
FUNCTION CB_dint_to_dword : DWORD

TITLE = ' Convert a double integer into an Dword '
VERSION : '1.0'
AUTHOR  : CB
NAME    : DinToDwo
FAMILY  : TNI

VAR_INPUT
    IN : DINT;
END_VAR

VAR_TEMP

END_VAR

BEGIN

CB_dint_to_dword := DINT_TO_DWORD(IN);

END_FUNCTION
